TYPE ST_FanucRobotGeneralCtrl :
STRUCT
	Command : ST_FanucRobot_CSharpCommand;
	Status : ST_FanucRobot_CSharpStatus;
END_STRUCT
END_TYPE

(* stored: Version 1.1.0.1, ProductVersion 3.1.4024.13
   DUT ST_FanucRobotGeneralCtrl: Id {4863966d-1047-4b37-84bb-5b6e908bf94e} *)
